INTERFACE I_Serializable EXTENDS __SYSTEM.IQueryInterface

METHOD SerializeWith
VAR_INPUT
	Serializer : I_Serializer;
END_VAR
END_METHOD

END_INTERFACE

(* stored: Version 1.1.0.1, ProductVersion 3.1.4024.12
   Itf I_Serializable: Id {17b600c5-ab7b-4b18-a049-defe2038de4c}
   Method SerializeWith: Id {5e384843-bd6d-4596-9678-cdd5191d1928} *)
